(* CoDeSys 2.3.9.37 project: Cap8_3_Res.pro *)
(* Libraries: Standard.lib 4.10.05 12:14:46 *)

(* Global variable list: Global_Variables *)
VAR_GLOBAL
     (* Entradas *)
     Habilita:BOOL;
    (* Salidas *)
     Verde:BOOL;
     Ambar:BOOL;
     Rojo:BOOL;
END_VAR

(* POU PLC_PRG, LD *)
PROGRAM PLC_PRG
VAR
         TempoRojo:TON;
        TempoAmbar:TON;
        TempoVerde:TON;
	FinVerde: BOOL;
	FinAmbar: BOOL;
	FinRojo: BOOL;
END_VAR
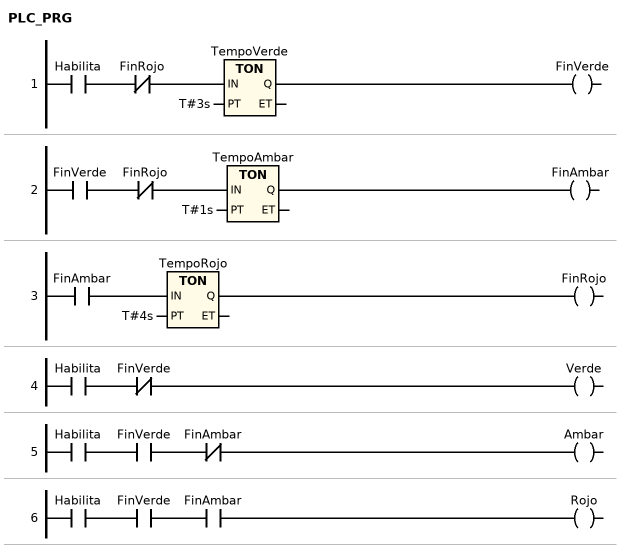
_LD_ (* Ladder Diagram *)
NETWORK 1
	[Habilita] - [/FinRojo] - TempoVerde:TON(IN: *, PT: T#3s) --- (FinVerde)
NETWORK 2
	[FinVerde] - [/FinRojo] - TempoAmbar:TON(IN: *, PT: T#1s) --- (FinAmbar)
NETWORK 3
	[FinAmbar] - TempoRojo:TON(IN: *, PT: T#4s) --- (FinRojo)
NETWORK 4
	[Habilita] - [/FinVerde] --- (Verde)
NETWORK 5
	[Habilita] - [FinVerde] - [/FinAmbar] --- (Ambar)
NETWORK 6
	[Habilita] - [FinVerde] - [FinAmbar] --- (Rojo)
_END_LD_
(* the same logic as Structured Text *)
(* Network 1 *)
TempoVerde(IN := Habilita AND NOT FinRojo, PT := T#3s);
FinVerde := TempoVerde.Q;
(* Network 2 *)
TempoAmbar(IN := FinVerde AND NOT FinRojo, PT := T#1s);
FinAmbar := TempoAmbar.Q;
(* Network 3 *)
TempoRojo(IN := FinAmbar, PT := T#4s);
FinRojo := TempoRojo.Q;
(* Network 4 *)
Verde := Habilita AND NOT FinVerde;
(* Network 5 *)
Ambar := Habilita AND FinVerde AND NOT FinAmbar;
(* Network 6 *)
Rojo := Habilita AND FinVerde AND FinAmbar;
END_PROGRAM

(* Visualisation Visu
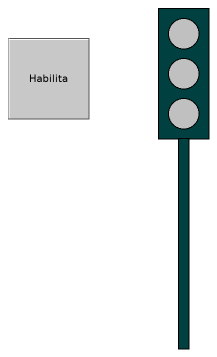
button at (20,50)-(101,131): text "Habilita"; toggles Habilita
ellipse at (180,30)-(211,61): alarm colour if Rojo
ellipse at (180,70)-(211,101): alarm colour if Ambar
ellipse at (180,110)-(211,141): alarm colour if Verde
2 more shapes without text or variables
*)
